FUNCTION_BLOCK FB_Chamber1SpinAxisMoveVelCWServices EXTENDS FB_ServiceBase
VAR_INPUT
	Param : ST_Chamber1SpinAxisMoveVelParam;
	Axis_BaseUnit : I_Axis_BaseUnit;
END_VAR

VAR
	_LatchedParam : ST_Chamber1SpinAxisMoveVelParam;
END_VAR

M_UpdateService(CompletionBehavior := E_ServiceCompletionBehavior.NaturalCompletion);

METHOD PROTECTED H_OnAborted
VAR_INPUT
	bFirstScan	: BOOL;
END_VAR
// Release defensively in case an unexpected transition skipped cleanup.
Axis_BaseUnit.M_ReleaseResource(OwnerId := ServiceId);
END_METHOD

METHOD PROTECTED H_OnAborting : E_PackMLHookResult
VAR_INPUT
	bFirstScan	: BOOL;
END_VAR

VAR
	bDone : BOOL;
	bError : BOOL;
	nErrorId : UDINT;
END_VAR
H_OnAborting := E_PackMLHookResult.Busy;

// A Service that never acquired the Resource must not reset its Owner's Axis.
IF NOT Axis_BaseUnit.M_IsResourceOwner(OwnerId := ServiceId) THEN
	H_OnAborting := E_PackMLHookResult.Done;
	RETURN;
END_IF

// Withdraw MoveVelocity before resetting the Axis.
Axis_BaseUnit.M_MoveVel(
	OwnerId := ServiceId,
	Execute := FALSE,
	Direction := MC_Direction.MC_Positive_Direction,
	Velocity := _LatchedParam.Velocity,
	Acceleration := _LatchedParam.Acceleration,
	Deceleration := _LatchedParam.Deceleration);
	
Axis_BaseUnit.M_Reset(
	OwnerId := ServiceId,
	Execute := TRUE,
	Done=> bDone, Error=> bError, ErrorId=> nErrorId);

IF bDone THEN
	Axis_BaseUnit.M_Reset(
		OwnerId := ServiceId,
		Execute := FALSE);
	// Keep ownership until the asynchronous Reset has completed.
	Axis_BaseUnit.M_ReleaseResource(OwnerId := ServiceId);
	H_OnAborting := E_PackMLHookResult.Done;

ELSIF bError THEN
	// A failed Reset is terminal for this Abort sequence; do not remain in Aborting.
	Axis_BaseUnit.M_Reset(
		OwnerId := ServiceId,
		Execute := FALSE);
	M_AddError(
		MainErrorId := E_Chamber1ErrorCode.Error_While_Reset_Axis,
		SourceErrorId := nErrorId,
		Message := 'Axis reset failed while aborting.');
	Axis_BaseUnit.M_ReleaseResource(OwnerId := ServiceId);
	H_OnAborting := E_PackMLHookResult.Done;
END_IF
END_METHOD

METHOD PROTECTED H_OnClearing : E_PackMLHookResult
VAR_INPUT
	bFirstScan	: BOOL;
END_VAR

VAR
	bServoOn : BOOL;
	bError : BOOL;
	nErrorId : UDINT;
END_VAR
H_OnClearing := E_PackMLHookResult.Done;
END_METHOD

METHOD PROTECTED H_OnComplete
VAR_INPUT
	bFirstScan	: BOOL;
END_VAR
// Reaching Complete means target velocity was reached; the Axis is still moving,
// so this Service must retain ownership until Stop or Abort cleanup finishes.
END_METHOD

METHOD PROTECTED H_OnCompleting : E_PackMLHookResult
VAR_INPUT
	bFirstScan	: BOOL;
END_VAR
Axis_BaseUnit.M_MoveVel(
	OwnerId := ServiceId,
	Execute := FALSE,
	Direction := MC_Direction.MC_Positive_Direction,
	Velocity := _LatchedParam.Velocity,
	Acceleration := _LatchedParam.Acceleration,
	Deceleration := _LatchedParam.Deceleration);

// Lowering Execute only withdraws the FB request; it does not stop the Axis.
// Keep ownership so a later Stop from Complete or Idle can control the motion.
H_OnCompleting := E_PackMLHookResult.Done;
END_METHOD

METHOD PROTECTED H_OnExecute : E_PackMLHookResult
VAR_INPUT
	bFirstScan	: BOOL;
END_VAR

VAR
	bInVelocity : BOOL;
	bError : BOOL;
END_VAR
H_OnExecute := E_PackMLHookResult.Busy;

// The Start-time snapshot remains fixed for the entire Execute phase.
Axis_BaseUnit.M_MoveVel(
	OwnerId := ServiceId,
	Execute := TRUE,
	Direction := MC_Direction.MC_Positive_Direction,
	Velocity := _LatchedParam.Velocity,
	Acceleration := _LatchedParam.Acceleration,
	Deceleration := _LatchedParam.Deceleration,
	InVelocity => bInVelocity,
	Error => bError);

IF bError THEN
	M_AddError(MainErrorId := E_Chamber1ErrorCode.Axis_Command_Error_During_Execute, SourceErrorId := 0, Message := 'MoveVelocity failed during Execute.');
	RequestCommand(E_PackMLCommand.Stop);
	RETURN;
END_IF

IF bInVelocity THEN
	H_OnExecute := E_PackMLHookResult.Done;
END_IF
END_METHOD

METHOD PROTECTED H_OnHeld
VAR_INPUT
	bFirstScan	: BOOL;
END_VAR
// Default action hook intentionally empty. Override in derived FBs when needed.
END_METHOD

METHOD PROTECTED H_OnHolding : E_PackMLHookResult
VAR_INPUT
	bFirstScan	: BOOL;
END_VAR
// Default transient hooks complete immediately; override when work is required.
H_OnHolding := E_PackMLHookResult.Done;
END_METHOD

METHOD PROTECTED H_OnIdle
VAR_INPUT
	bFirstScan	: BOOL;
END_VAR
// Reset changes only the PackML state. A MoveVel that completed naturally may
// still be moving, so Idle intentionally retains any existing Axis ownership.
END_METHOD

METHOD PROTECTED H_OnResetting : E_PackMLHookResult
VAR_INPUT
	bFirstScan	: BOOL;
END_VAR
MEMSET(ADR(Status.ErrorList), 0, SIZEOF(Status.ErrorList));

H_OnResetting := E_PackMLHookResult.Done;
END_METHOD

METHOD PROTECTED H_OnStarting : E_PackMLHookResult
VAR_INPUT
	bFirstScan	: BOOL;
END_VAR
H_OnStarting := E_PackMLHookResult.Busy;

// Validate Service-owned data before reserving the shared BaseUnit.
IF Param.Velocity <= 0 THEN
	M_AddError(MainErrorId := E_Chamber1ErrorCode.Invalid_Param, SourceErrorId := 0, Message := 'Velocity must be greater than zero.');
	RequestCommand(E_PackMLCommand.Stop);
	RETURN;
END_IF

IF Param.Acceleration < 0 THEN
	M_AddError(MainErrorId := E_Chamber1ErrorCode.Invalid_Param, SourceErrorId := 0, Message := 'Acceleration must not be negative.');
	RequestCommand(E_PackMLCommand.Stop);
	RETURN;
END_IF

IF Param.Deceleration < 0 THEN
	M_AddError(MainErrorId := E_Chamber1ErrorCode.Invalid_Param, SourceErrorId := 0, Message := 'Deceleration must not be negative.');
	RequestCommand(E_PackMLCommand.Stop);
	RETURN;
END_IF

// Keep one fixed command snapshot until the Service leaves this run.
_LatchedParam := Param;

// Resource contention is a failed Start, not a wait condition.
IF NOT Axis_BaseUnit.M_AcquireResource(OwnerId := ServiceId) THEN
	M_AddError(MainErrorId := E_Chamber1ErrorCode.Resource_Acquire_Failed_During_Starting, SourceErrorId := 0, Message := 'Axis resource acquisition failed during Starting.');
	RequestCommand(E_PackMLCommand.Stop);
	RETURN;
END_IF

// Physical checks occur only after this Service owns the BaseUnit.
IF Axis_BaseUnit.AxisIsDisabled THEN
	M_AddError(MainErrorId := E_Chamber1ErrorCode.Axis_Not_Servo_On_During_Starting, SourceErrorId := 0, Message := 'Axis is not servo on during Starting.');
	RequestCommand(E_PackMLCommand.Abort);
	RETURN;
END_IF

IF Axis_BaseUnit.AxisHasJob THEN
	M_AddError(MainErrorId := E_Chamber1ErrorCode.Axis_Is_Busy_During_Starting, SourceErrorId := 0, Message := 'Axis is busy during Starting.');
	RequestCommand(E_PackMLCommand.Stop);
	RETURN;
END_IF

H_OnStarting := E_PackMLHookResult.Done;
END_METHOD

METHOD PROTECTED H_OnStopped
VAR_INPUT
	bFirstScan	: BOOL;
END_VAR
// Release defensively after every Stop path.
Axis_BaseUnit.M_ReleaseResource(OwnerId := ServiceId);
END_METHOD

METHOD PROTECTED H_OnStopping : E_PackMLHookResult
VAR_INPUT
	bFirstScan	: BOOL;
END_VAR

VAR
	bDone : BOOL;
	bError : BOOL;
	nErrorId : UDINT;
END_VAR
H_OnStopping := E_PackMLHookResult.Busy;

// Resource acquisition failures enter Stopping without owning the Axis.
IF NOT Axis_BaseUnit.M_IsResourceOwner(OwnerId := ServiceId) THEN
	H_OnStopping := E_PackMLHookResult.Done;
	RETURN;
END_IF

// Withdraw MoveVelocity before issuing the physical Stop.
Axis_BaseUnit.M_MoveVel(
	OwnerId := ServiceId,
	Execute := FALSE,
	Direction := MC_Direction.MC_Positive_Direction,
	Velocity := _LatchedParam.Velocity,
	Acceleration := _LatchedParam.Acceleration,
	Deceleration := _LatchedParam.Deceleration);
	
Axis_BaseUnit.M_Stop(
	OwnerId := ServiceId,
	Execute := TRUE, 
	Deceleration:= _LatchedParam.Deceleration,
	Done=> bDone, Error=> bError, ErrorId=> nErrorId);

IF bDone THEN
	Axis_BaseUnit.M_Stop(
		OwnerId := ServiceId,
		Execute := FALSE, 
		Deceleration:= _LatchedParam.Deceleration);
	// Ownership is released only after the asynchronous Stop has completed.
	Axis_BaseUnit.M_ReleaseResource(OwnerId := ServiceId);
	H_OnStopping := E_PackMLHookResult.Done;
	
ELSIF bError THEN
	// Throw up error
	M_AddError(
		MainErrorId := E_Chamber1ErrorCode.Error_While_Stop_Axis,
		SourceErrorId := nErrorId,
		Message := 'Axis stop failed while stopping.');
	
	Axis_BaseUnit.M_Stop(
		OwnerId := ServiceId,
		Execute := FALSE, 
		Deceleration:= _LatchedParam.Deceleration);
		
	RequestCommand(E_PackMLCommand.Abort);
END_IF
END_METHOD

METHOD PROTECTED H_OnSuspended
VAR_INPUT
	bFirstScan	: BOOL;
END_VAR
// Default action hook intentionally empty. Override in derived FBs when needed.
END_METHOD

METHOD PROTECTED H_OnSuspending : E_PackMLHookResult
VAR_INPUT
	bFirstScan	: BOOL;
END_VAR
// Default transient hooks complete immediately; override when work is required.
H_OnSuspending := E_PackMLHookResult.Done;
END_METHOD

METHOD PROTECTED H_OnUndefined : E_PackMLHookResult
VAR_INPUT
	bFirstScan	: BOOL;
END_VAR
// The base FB leaves Undefined immediately unless a derived FB delays startup.
H_OnUndefined := E_PackMLHookResult.Done;
END_METHOD

METHOD PROTECTED H_OnUnholding : E_PackMLHookResult
VAR_INPUT
	bFirstScan	: BOOL;
END_VAR
// Default transient hooks complete immediately; override when work is required.
H_OnUnholding := E_PackMLHookResult.Done;
END_METHOD

METHOD PROTECTED H_OnUnsuspending : E_PackMLHookResult
VAR_INPUT
	bFirstScan	: BOOL;
END_VAR
// Default transient hooks complete immediately; override when work is required.
H_OnUnsuspending := E_PackMLHookResult.Done;
END_METHOD

END_FUNCTION_BLOCK

(* stored: Version 1.1.0.1, ProductVersion 3.1.4026.18
   POU FB_Chamber1SpinAxisMoveVelCWServices: Id {2d3a48e0-0a65-435f-812d-3e25cfaffe3c}, SpecialFunc None
   Folder StateAction: Id {49ed7549-95d2-4542-8c09-83ad057d2672}
   Method H_OnAborted: Id {328f5265-3f48-4442-8390-1fd00d156006}
   Method H_OnAborting: Id {8ef4724f-e418-45d4-b245-336c28b5f1de}
   Method H_OnClearing: Id {e065280f-e16e-4d87-85cf-24b54094afe6}
   Method H_OnComplete: Id {6d77d87d-d9c6-4390-a07a-5b4202d501b8}
   Method H_OnCompleting: Id {3864e1ba-9360-45a8-9d26-f1e180c8fbe5}
   Method H_OnExecute: Id {d5c34347-be90-4f5e-8be4-57798b5c5bb2}
   Method H_OnHeld: Id {290e557c-077d-4d3a-a2bb-06d511e35f5d}
   Method H_OnHolding: Id {fa63c046-0d26-4f2c-83a5-fda321bd6ee0}
   Method H_OnIdle: Id {59828899-47c9-4777-90f1-23e06ffd978a}
   Method H_OnResetting: Id {0680bc64-d1f9-407b-b6ca-83882b900618}
   Method H_OnStarting: Id {ce6c9548-1f79-4b75-96e2-343a2f8f84cb}
   Method H_OnStopped: Id {768434f7-cc85-4fdb-a507-f054649262b4}
   Method H_OnStopping: Id {b2816703-e998-4497-a19c-1d20e18f1f4c}
   Method H_OnSuspended: Id {3237239b-48f7-46dc-b2a0-07f7727d1af4}
   Method H_OnSuspending: Id {21d2483c-a2c4-4efb-8137-575165e782fc}
   Method H_OnUndefined: Id {355660e6-63b3-47e1-98ff-81122ad86689}
   Method H_OnUnholding: Id {4d791b75-be71-409c-890a-fcf31649efc0}
   Method H_OnUnsuspending: Id {cd52fade-963d-45ca-a66e-acbc7e8b9c95} *)
